{attribute addProperty BoxType "KL2284"}
{attribute addProperty Id "CWAT %Q*BOOL000CCWAT %Q*BOOL000"}
{attribute addProperty CRC "2651204892"}
{attribute addProperty SizeInBites "0"}
{attribute addProperty SizeInBytes "0"}
TYPE Channel_9E062D1C :
STRUCT
	{attribute addProperty Name "CW"}
	CW AT %Q* : BOOL;
	{attribute addProperty Name "CCW"}
	CCW AT %Q* : BOOL;
END_STRUCT
END_TYPE

(* stored: Version 1.2.0.0, ProductVersion 3.1.4024.9
   DUT Channel_9E062D1C: Id {e805305b-13ea-45cd-b199-c518efc63cba} *)
